Staubli VAL3: remErrNum.pgx

program remErrNum(string sCmd (dimensions=1), string& sArg[] (dimensions=1), string& sReturn[] (dimensions=1))
begin
  // Error raised when we recieve an non-numerical argument when
  // a number was expected.
  //
  logMsg("call remErrNum")
  sReturn="ERROR 103: "+sCmd+"non-num arg '"+sArg+"'"
  putln(sReturn)
  logMsg(sReturn)
end
